// TIA Portal V19 export
TYPE "LUC_typeSignalStackByDInt"
// Stack Light Signals by DINT
// stored: Access Published
   STRUCT
      red { ExternalWritable := 'False'} : DInt;   // Red light active
      yellow { ExternalWritable := 'False'} : DInt;   // Yellow light active
      blue { ExternalWritable := 'False'} : DInt;   // Blue light active
      green { ExternalWritable := 'False'} : DInt;   // Green light active
      horn { ExternalWritable := 'False'} : DInt;   // Horn active
      white { ExternalWritable := 'False'} : DInt;   // White light active
      user1 { ExternalWritable := 'False'} : DInt;   // User defined light 1 active
      user2 { ExternalWritable := 'False'} : DInt;   // User defined light 2 active
   END_STRUCT;
END_TYPE
